(* IEC 61131-3 sources: CodesysTest/alpha/export/FBs/Components/Load Plate/FB_BaseLoadPlate.pou/Internal/LoadPlateToDischarge.prop, 1 file *)

(* ---- Get.pm.st ---- *)
(*#-#-#-#-#-#-#-#-#-#---Declaration---#-#-#-#-#-#-#-#-#-#-#-#-#*)

VAR
END_VAR
(*#-#-#-#-#-#-#-#-#-#---Implementation---#-#-#-#-#-#-#-#-#-#-#-#-#*)

LoadPlateToDischarge := _manualOn OR ((_triggerActiveONS.OSR OR _shakeActiveONS.OSF) AND inUse) OR ((_estopOK.OSR OR _disabledPositionHasUpdated OR _loadPlateInUseONS.OSF) AND disabledPosition = PackageEjectionDisabledPosition.DischargePosition AND NOT inUse);
